(* IEC 61131-3 sources: programs/VI-54/VI-54_20171205/VI-54_20171205/Stations/Screen/LseClass170718/Class/inpLine, 1 file *)

(* ---- inpLine.st ---- *)
(*!
<Class
	Name               = "inpLine"
	Revision           = "0.0"
	RealtimeTask       = "false"
	CyclicTask         = "false"
	BackgroundTask     = "false"
	Sigmatek           = "false"
	OSInterface        = "false"
	HighPriority       = "false"
	Automatic          = "false"
	UpdateMode         = "Prescan"
	SharedCommandTable = "true"
	Objectsize         = "(840,960)">
	<Channels>
		<Server Name="_______________" Visualized="false" Initialize="false" WriteProtected="true" Retentive="false"/>
		<Server Name="LineSpeed" Visualized="true" Initialize="false" WriteProtected="false" Retentive="false"/>
		<Server Name="MaxAccDecInfeedConv" Visualized="true" Initialize="false" WriteProtected="true" Retentive="false"/>
		<Server Name="MaxSpeedInfeedConv" Visualized="true" Initialize="false" WriteProtected="true" Retentive="false"/>
		<Server Name="TrayLenght" Visualized="false" Initialize="false" WriteProtected="false" Retentive="false"/>
		<Server Name="TraysPerMinute" Visualized="true" Initialize="false" WriteProtected="false" Retentive="false"/>
	</Channels>
	<Network Name="inpLine">
		<!-- List of Components in this network -->
		<Components>
			<Object
				Name       = "_base"
				Class      = "ReceptBase"
				Position   = "(218,120)"
				Visualized = "false">
				<Channels>
					<Server Name="Refresh"/>
					<Server Name="Size"/>
					<Client Name="Data"/>
				</Channels>
			</Object>
		</Components>
		<Comments>
		</Comments>
		<!-- List of Connections in this network -->
		<Connections>
			<Connection Source="this.Refresh" Destination="_base.Refresh" Vertices="(690,210),(518,210),"/>
			<Connection Source="this.Size" Destination="_base.Size" Vertices="(690,270),(518,270),"/>
			<Connection Source="_base.Data" Destination="this.Data" Vertices="(218,210),(38,210),"/>
		</Connections>
		<!-- Headerfiles -->
		<Options>
		</Options>
	</Network>
</Class>
*)
#pragma using ReceptBase

inpLine : CLASS
: ReceptBase
  //Servers:
	MaxSpeedInfeedConv 	: SvrCh_DINT;
	MaxAccDecInfeedConv 	: SvrCh_DINT;
	_______________ 	: SvrCh_DINT;
	LineSpeed 	: SvrCh_DINT;
	TraysPerMinute 	: SvrCh_DINT;
	TrayLenght 	: SvrCh_DINT;
  //Clients:
  //Variables:
  //Functions:

	FUNCTION VIRTUAL GLOBAL Init;

	FUNCTION VIRTUAL GLOBAL DefaultPara;

	FUNCTION VIRTUAL GLOBAL RefreshPara;

	FUNCTION VIRTUAL GLOBAL LineSpeed::Write
		VAR_INPUT
			input (EAX) 	: DINT;
		END_VAR
		VAR_OUTPUT
			result (EAX) 	: DINT;
		END_VAR;

	FUNCTION VIRTUAL GLOBAL TraysPerMinute::Write
		VAR_INPUT
			input (EAX) 	: DINT;
		END_VAR
		VAR_OUTPUT
			result (EAX) 	: DINT;
		END_VAR;

	FUNCTION VIRTUAL GLOBAL TrayLenght::Write
		VAR_INPUT
			input (EAX) 	: DINT;
		END_VAR
		VAR_OUTPUT
			result (EAX) 	: DINT;
		END_VAR;
  //Tables:
	FUNCTION @STD
		VAR_OUTPUT
			ret_code	: CONFSTATES;
		END_VAR;
	FUNCTION GLOBAL TAB @CT_;
END_CLASS;

FUNCTION VIRTUAL GLOBAL inpLine::Init

  //MaxSpeedInfeedConv  := to_dint(to_real cInfeedConvVmax95proc ToMperMin);
  //MaxAccDecInfeedConv := to_dint(to_real cInfeedConvAmax ToMperSec2);

  // Call init from receptbase
  ReceptBase::Init();

END_FUNCTION

FUNCTION VIRTUAL GLOBAL inpLine::DefaultPara

END_FUNCTION

FUNCTION VIRTUAL GLOBAL inpLine::RefreshPara

  ReceptPtr^.Machine.TraysPerMinute          := TraysPerMinute;
  ReceptPtr^.Machine.TrayLenght              := TrayLenght;

END_FUNCTION

FUNCTION VIRTUAL GLOBAL inpLine::TraysPerMinute::Write
	VAR_INPUT
		input (EAX) 	: DINT;
	END_VAR
	VAR_OUTPUT
		result (EAX) 	: DINT;
	END_VAR

	TraysPerMinute := input;
  ReceptPtr^.Machine.TraysPerMinute := TraysPerMinute;
	result := TraysPerMinute;

END_FUNCTION

FUNCTION VIRTUAL GLOBAL inpLine::TrayLenght::Write
	VAR_INPUT
		input (EAX) 	: DINT;
	END_VAR
	VAR_OUTPUT
		result (EAX) 	: DINT;
	END_VAR

	TrayLenght := input;
  ReceptPtr^.Machine.TrayLenght := TrayLenght;
	result := TrayLenght;

END_FUNCTION

FUNCTION VIRTUAL GLOBAL inpLine::LineSpeed::Write
	VAR_INPUT
		input (EAX) 	: DINT;
	END_VAR
	VAR_OUTPUT
		result (EAX) 	: DINT;
	END_VAR

	LineSpeed := input;
  ReceptPtr^.Machine.LineSpeed := LineSpeed;
	result := LineSpeed;

END_FUNCTION
